// TIA Portal V20 export
TYPE "UDT_POS_AXES_UVW"
   STRUCT
      U_POS_EXTERNAL_LOAD : Real;
      U_POS_EXTERNAL_UNLOAD : Real;
      U_POS_SAS : Real;
      U_POS_BLOWING : Real;
      U_POS_DETECTOR_LOAD : Real;
      U_POS_DETECTOR_UNLOAD : Real;
      U_POS_INTERNAL_LOADER_LOAD : Real;
      U_POS_INTERNAL_LOADER_UNLOAD : Real;
      U_POS_OUT_INTERNAL_LOADER : Real;
      U_DELTA_POS_INTERN_LOADER_LOAD_UNLOAD : Real;
      U_POS_SEMI_AUTO : Real;
      V_POS_SHUTTLE_LOAD : Real;
      V_POS_SHUTTLE_UNLOAD : Real;
      V_POS_WASHING : Real;
      W_POS_UP : Real;
      W_POS_SHUTTLE_LOAD : Real;
      W_POS_SHUTTLE_UNLOAD : Real;
      W_POS_WASHING : Real;
      X_POS_CHANGE_BW : Real;
      Y_POS_CHANGE_BW : Real;
   END_STRUCT;
END_TYPE
